// TIA Portal V18 export
VAR_GLOBAL   // PLC tag table "Default tag table_1"
   qw100_1 AT %QW100 : Word;
   iw0_1 AT %IW0 : Word;
   qw0 AT %QW0 : Word;
   iw500_1 AT %IW500 : Word;
   qw500_1 AT %QW500 : Word;
   iw100_1 AT %IW100 : Word;
   qw600_1 AT %QW600 : Word;
   iw102_3 AT %IW102 : Word;
   qw602_3 AT %QW602 : Word;
   iw600_1 AT %IW600 : Word;
   iw602_3 AT %IW602 : Word;
   w102_3 AT %QW102 : Word;
   di_800 AT %ID800 : DWord;
   di_801 AT %ID804 : DWord;
   di_802 AT %ID808 : DWord;
   di_803 AT %ID812 : DWord;
   di_804 AT %ID816 : DWord;
   di_805 AT %ID820 : DWord;
   di_806na AT %ID824 : DWord;
   vdq700 AT %QD700 : DWord;
   vdq701 AT %QD704 : DWord;
   vdq702 AT %QD708 : DWord;
   vdq703 AT %QD712 : DWord;
   vdq704 AT %QD716 : DWord;
   vdq705 AT %QD720 : DWord;
   vdq706na AT %QD724 : DWord;
   dq800 AT %QD800 : DWord;
   dq801 AT %QD804 : DWord;
   dq802 AT %QD808 : DWord;
   dq803 AT %QD812 : DWord;
   dq804 AT %QD816 : DWord;
   dq805 AT %QD820 : DWord;
   dq806na AT %QD824 : DWord;
   vdi700 AT %ID700 : DWord;
   vdi701 AT %ID704 : DWord;
   vdi702 AT %ID708 : DWord;
   vdi703 AT %ID712 : DWord;
   vdi704 AT %ID716 : DWord;
   vdi705 AT %ID720 : DWord;
   vdi706na AT %ID724 : DWord;
   commiw_50 AT %IW50 : Word;
   commqw_50 AT %QW50 : Word;
   Connection_lost AT %M0.0 : Bool;
   mem AT %MW2 : Word;
END_VAR
VAR_GLOBAL CONSTANT   // user constants
   "None(1)" : Pip := 65535;
   "Automatic update(1)" : Pip := 0;
   "PIP 1(1)" : Pip := 1;
   "PIP 2(1)" : Pip := 2;
   "PIP 3(1)" : Pip := 3;
   "PIP 4(1)" : Pip := 4;
   "PIP OB Servo(1)" : Pip := 32768;
   "Local~MC(1)" : Hw_SubModule := 51;
   "Local~Exec(1)" : Hw_SubModule := 52;
   "Local(1)" : Hw_SubModule := 49;
   "Local~PROFINET_interface_1(1)" : Hw_Interface := 64;
   "Local~PROFINET_interface_1~Port_1(1)" : Hw_Interface := 65;
   "Local~PROFINET_interface_1~Port_2(1)" : Hw_Interface := 66;
   "Local~HSC_1(1)" : Hw_Hsc := 257;
   "Local~HSC_2(1)" : Hw_Hsc := 258;
   "Local~HSC_3(1)" : Hw_Hsc := 259;
   "Local~HSC_4(1)" : Hw_Hsc := 260;
   "Local~HSC_5(1)" : Hw_Hsc := 261;
   "Local~HSC_6(1)" : Hw_Hsc := 262;
   "Local~AI_2_AQ_2_1(1)" : Hw_SubModule := 263;
   "Local~DI_14_DQ_10_1(1)" : Hw_SubModule := 264;
   "Local~OPC_UA(1)" : Hw_SubModule := 117;
   "Local~Pulse_1(1)" : Hw_Pwm := 265;
   "Local~Pulse_2(1)" : Hw_Pwm := 266;
   "Local~Pulse_3(1)" : Hw_Pwm := 267;
   "Local~Pulse_4(1)" : Hw_Pwm := 268;
   "Local~PROFINET_interface_1~IODevice" : Hw_Device := 270;
   "Local~PROFINET_interface_1~bool0" : Hw_SubModule := 272;
   "Local~PROFINET_interface_1~bool1" : Hw_SubModule := 273;
   "Local~PROFINET_interface_1~analog0" : Hw_SubModule := 274;
   "Local~PROFINET_interface_1~anolog1" : Hw_SubModule := 275;
   "Local~PROFINET_interface_1~hsc" : Hw_SubModule := 276;
   "Local~PROFINET_interface_1~pulse" : Hw_SubModule := 277;
   "Local~PROFINET_interface_1~comm0" : Hw_SubModule := 278;
   "Local~PROFINET_interface_1~comm1" : Hw_SubModule := 279;
   "Local~Common(1)" : Hw_SubModule := 50;
   "Local~Device(1)" : Hw_Device := 32;
   "Local~Configuration(1)" : Hw_SubModule := 33;
   "OB_Cyclic interrupt(1)" : OB_Cyclic := 30;
END_VAR
